FUNCTION_BLOCK Test_TStreamAdd_Read_LREAL_CheckAlignment EXTENDS T_UnitTestBase
VAR
    Stream  : T_Stream(StreamLength := 2);
    ArgType : E_ArgTypeId := E_ArgTypeId.Type_LREAL;
END_VAR

METHOD  Init
VAR_INPUT
END_VAR
END_METHOD

{attribute 'analysis' := '-33'} // inhibit unused variable warning
METHOD RunTest
Stream.Init(2);

Stream.Add_BYTE(123);// add a byte to test alignment checks...
Stream.Add_LREAL(1.234567891234);

Stream.SetReadPosition(0);

Stream.Read_BYTE();

// check next value...	
AssertEquals_LREAL(Expected     := 1.234567891234,
                             Actual       := Stream.Read_LREAL(),
                             Delta        := 0.000000000001,
                             Message := 'Stream.Read_LREAL()');

// check we are at the end of the stream..							
AssertEquals_UDINT(Expected     := Stream.StreamLength,
                             Actual       := Stream.ReadPosition,
                             Message := 'Stream.ReadPosition');

TestCompleted := TRUE;
END_METHOD

END_FUNCTION_BLOCK

(* stored: Version 1.1.0.1, ProductVersion 3.1.4024.12
   POU Test_TStreamAdd_Read_LREAL_CheckAlignment: Id {24ee5d05-14c7-4334-b9cb-4c7dec7a4439}, SpecialFunc None
   Method Init: Id {800ce986-d6d3-4c98-b81c-be3b526ddffd}
   Method RunTest: Id {f98297ca-ab0f-4e0b-8756-bd55c1387389} *)
